FUNCTION_BLOCK TeknicHardWire_old //EXTENDS EncodedDrive
VAR_INPUT
	bEnable : BOOL;
END_VAR
VAR_OUTPUT
	enable AT %Q* : BOOL; //enable + pulses
	A AT %Q* : BOOL; //direction (F = inwards, T = outwards)
	B AT %Q* : BOOL; //home bit
	brakeRelease AT %Q* : BOOL;
	
	contact AT %I* : BOOL;
	
	home AT %I* : BOOL;
	outerLimit AT %I* : BOOL;
	innerLimit AT %I* : BOOL;
	
	homeSet : BOOL;
	busy : BOOL;
	error : BOOL;
	done AT %I* : BOOL;
	
	position : LREAL;
	targetPos : LREAL;
END_VAR
VAR
	pulseCounter : INT;
	pulser : TON;
	
	resetTimer : TP;
	
	mode : (HOLD, TARGET, CONTINUOUS);	
	step : Homing;//(IDLE, HOME_UP, HOME_FINAL, DOWN, REDO_HOME, HOME_DONE);
END_VAR
VAR_STAT CONSTANT
	resetPulseWidth : TIME := T#1000MS;
	pulseWidth : TIME := T#25MS;
	unitsPerPulse : INT := 800; //800 Teknic units per revolution
	distancePerPulse : INT := 5; //5mm per revolution
END_VAR

IF NOT bEnable THEN
	mode := HOLD;
END_IF

resetTimer(IN:= , PT:= resetPulseWidth, Q=> , ET=> );
IF resetTimer.Q THEN
	resetTimer.IN := FALSE;	
	mode := HOLD;
	//RETURN;
ELSIF resetTimer.IN THEN
	enable := FALSE;
	mode := HOLD;
	//RETURN;
END_IF


CASE mode OF
	HOLD:
		IF NOT resetTimer.IN THEN
			enable := bEnable;
		END_IF
		pulseCounter := 0;
	
	TARGET:
		(*
		//this block calculates the number of pulses beforehand using new position every cycle, may exceed travel limits
		//may not be suitable as the position is calculated up front and may exceed the actual travel limits
		IF WithinTolerance(position, target, unitsPerPulse) THEN
			pulseCounter := 0;
			mode := HOLD;
			
		ELSIF NOT busy THEN
			A := position < target;
			//requestPulses(1);
			requestPulses( TO_INT(CEILING(ABS(position - targetPos)/distancePerPulse)) );
		END_IF
		*)
		//(*
		//this block sends one pulse at a time until the target position is reached
		//positioning is more accurate but motion is choppy
		IF WithinTolerance(position, target, unitsPerPulse) THEN
			pulseCounter := 0;
			mode := HOLD;
		ELSIF NOT busy THEN
			A := position < target;
			requestPulses(1);
		END_IF
		//*)
	CONTINUOUS:
		requestPulses(1);
		
END_CASE

IF home OR innerLimit OR outerLimit THEN
	pulseCounter := 0;
	mode := HOLD;
END_IF

sequence();

METHOD homingSequence : BOOL
CASE step OF
	Homing.IDLE:
		enable := FALSE;
		A := FALSE;
		B := FALSE;
		brakeRelease := TRUE;
		
		homeSet := FALSE;
		step := Homing.REDO;
		
	Homing.REDO: //let insertion drop to inner limit before homing
		enable := FALSE;
		A := FALSE;
		B := FALSE;
		brakeRelease := TRUE;
		
		IF NOT innerLimit THEN
			enable := TRUE;
			step := Homing.HOME_OUT;
		END_IF
	
	Homing.HOME_OUT:
		enable := TRUE;
		A := FALSE;
		B := TRUE;
		brakeRelease := TRUE;
		
		IF NOT home THEN
			B := FALSE;
			step := Homing.DONE;
		END_IF
		
	Homing.DONE:
		//enable := FALSE;
		A := FALSE;
		B := FALSE;
		brakeRelease := TRUE;
		
		position := 0;
		homeSet := TRUE;
		homingSequence := TRUE;
		step := Homing.IDLE;
	
END_CASE
END_METHOD

METHOD moveAbsolute : BOOL
VAR_INPUT
	newTarget : LREAL;
END_VAR
targetPos := newTarget;
mode := TARGET;
END_METHOD

METHOD moveContinuous : BOOL
VAR_INPUT
	direction : MC_Direction;
END_VAR
IF direction = MC_Negative_Direction THEN
	A := FALSE;
ELSIF direction = MC_Positive_Direction THEN
	A := TRUE;
END_IF

mode := CONTINUOUS;
END_METHOD

METHOD PRIVATE requestPulses : BOOL
VAR_INPUT
	request : INT;
END_VAR
IF (done OR pulseCounter = 0) AND request > 0 THEN
	pulseCounter := request;
	
	requestPulses := TRUE;
END_IF
END_METHOD

METHOD reset : BOOL
VAR_INPUT
END_VAR
resetTimer.IN := TRUE;
END_METHOD

METHOD sequence : BOOL
VAR_INPUT
END_VAR
pulser(IN:= , PT:= pulseWidth, Q=> , ET=> ); //when timer is enabled, this toggles enable every <pulseWidth>

IF pulseCounter = 0 THEN
	busy := FALSE;
	
	enable := TRUE;
	pulser.IN := FALSE;
	RETURN;
END_IF

busy := TRUE;
pulser.IN := TRUE;

IF pulser.Q THEN
	pulser.IN := FALSE;
	enable := NOT enable;
	
	IF enable THEN //enable is TRUE after toggle
		pulseCounter := pulseCounter - 1;
		
		IF A THEN
			position := position + distancePerPulse;
		ELSE
			position := position - distancePerPulse;
		END_IF
	END_IF
	
END_IF
END_METHOD

METHOD stop : BOOL
VAR_INPUT
END_VAR
mode := HOLD;
END_METHOD

END_FUNCTION_BLOCK

(* stored: Version 1.1.0.1, ProductVersion 3.1.4024.11
   POU TeknicHardWire_old: Id {f2f2a1c1-ef3e-4af6-9287-f7b73dfedc95}, SpecialFunc None
   Method homingSequence: Id {4c078f6b-5e30-4406-b11a-fba70e03b84b}
   Method moveAbsolute: Id {de1b0ff3-ba6a-4c46-b761-cdd04c29ba51}
   Method moveContinuous: Id {2d54b74f-51c6-4f44-aa9a-a0185ebc66f6}
   Method requestPulses: Id {9be2f5f0-4c2c-424d-a26b-bcf77a93b753}
   Method reset: Id {1c45bc6e-39b8-4809-b9a5-c28ef542dac2}
   Method sequence: Id {2ad1a8af-5aed-432e-8bcf-5e2ff870d8fe}
   Method stop: Id {3a72c02a-16d6-478a-94db-f93b53410a9a} *)
